PROGRAM P_BACnet_Alarm
VAR
END_VAR

//keep BACnet object instance alive
fbBACnet_BV_Alarm(Device := Device, bEnablePV := TRUE, bNullPV := FALSE);

END_PROGRAM

(* stored: Version 1.1.0.1, ProductVersion 3.1.4024.5
   POU P_BACnet_Alarm: Id {11efe370-1957-4d2f-93d6-f1cebaa90845}, SpecialFunc None *)
